// TIA Portal project "Ex1-TheCraneProject" (V16)

(* hardware
DEVICE "S7-1200 station_1"  S7-1200 Station
   slot 0: "Rack_0"  S7-1200 Rack  Rack  V1.0
   slot 1: "PLC_1"  CPU 1215C DC/DC/Rly  6ES7 215-1HG40-0XB0  V4.4
   slot 101: "CM 1243-5"  CM 1243-5  6GK7 243-5DX30-0XE0  V1.3
DEVICE "GSD device_1"  GSD.Device
   slot 0: "Rack_0"  Rail
DEVICE "GSD device_2"  GSD.Device
   slot 0: "Rack_0"  Rail
DEVICE "GSD device_3"  GSD.Device.PN
   slot 0: "Rack"  Rack  V1.0
   slot 0: "cx8093"  CX8093 Profinet IO  Device V2.3, 2 Port  CX8093  V1.00
      slot 0: "CX8093 Profinet IO  Device V2.3, 2 Port_1"  CX8093 Profinet IO  Device V2.3, 2 Port
      slot 1: "CX8093 Profinet IO  Device V2.3, 2 Port"  CX8093 Profinet IO  Device V2.3, 2 Port
         slot 1: "Port 1"  Port 1
         slot 2: "Port 2"  Port 2
   slot 1: "1 Byte Input_1"  1 Byte Input
      slot 0: "1 Byte Input"  1 Byte Input
DEVICE "GSD device_4"  GSD.Device.PN
   slot 0: "Rack"  Rack  V1.0
   slot 0: "SI-PROFINET"  Commander C200-C300  SI-PROFINET
      slot 0: "Commander C200-C300"  Commander C200-C300
      slot 1: "X1"  X1
         slot 1: "X1 P1"  X1 P1
         slot 2: "X1 P2"  X1 P2
DEVICE "ET 200S station_1"  ET 200S station
   slot 0: "Rack_0"  Rail
   slot 0: "IO device_1"  IM 151-3 PN FO  6ES7 151-3BB23-0AB0  V7.0
   slot 1: "PM-E DC24V HF_1"  PM-E DC24V HF  6ES7 138-4CA60-0AB0
   slot 2: "2AI x U HF_1"  2AI x U HF  6ES7 134-4LB02-0AB0
   slot 3: "PM-D 24VDC_1"  PM-D 24VDC  3RK1 903-0BA00
   slot 4: "DSS1e-x HF 0,3-3A_1"  DSS1e-x HF 0,3-3A  3RK1 301-0AB20-0AB4  V10.0
   slot 5: "DSS1e-x HF 0,3-3A_2"  DSS1e-x HF 0,3-3A  3RK1 301-0AB20-0AB4  V10.0
   slot 6: "DSS1e-x HF 0,3-3A_3"  DSS1e-x HF 0,3-3A  3RK1 301-0AB20-0AB4  V10.0
*)

// ===== PLC "PLC_1"  CPU 1215C DC/DC/Rly =====

VAR_GLOBAL   // PLC tag table "Default tag table"
   "iBtnStart" AT %I0.0 : Bool;
   "iBtnStop" AT %I0.1 : Bool;
   "iBtnReset" AT %I0.2 : Bool;
   "iBtnEms" AT %I0.3 : Bool;
   "qLedStart" AT %Q0.0 : Bool;
   "qLedError" AT %Q0.1 : Bool;
END_VAR

ORGANIZATION_BLOCK "Main"   // OB1, LAD, ProgramCycle
TITLE = "Main Program Sweep (Cycle)"
{ S7_Optimized_Access := 'TRUE' }
VERSION : 0.1
   VAR_INPUT
      Initial_Call : Bool;   // Initial call of this OB
      Remanence : Bool;   // =True, if remanent data are available
   END_VAR
BEGIN
END_ORGANIZATION_BLOCK